INTERFACE Iterator

METHOD current : Object
VAR_INPUT
END_VAR
END_METHOD

METHOD hasNext : BOOL
VAR_INPUT
END_VAR
END_METHOD

METHOD next : Object
VAR_INPUT
END_VAR
END_METHOD

PROPERTY Position : INT
GET
END_GET
END_PROPERTY

METHOD reset : BOOL
VAR_INPUT
END_VAR
END_METHOD

END_INTERFACE

(* stored: Version 1.1.0.1, ProductVersion 3.1.4024.12
   Itf Iterator: Id {11e57a1b-5b87-41c6-8866-dab19c5cc778}
   Method current: Id {d60b1888-45a1-4719-b843-c166d488b64a}
   Method hasNext: Id {6e2d7f23-86d9-421b-a328-b7469453c32f}
   Method next: Id {a0f9df8b-6678-45f8-a11d-40ecbf79b0f8}
   Property Position: Id {b2d58fb3-5dc1-4b10-b185-0b3038c26065}
   Get Get: Id {35a09d46-efa2-4701-858c-533b3fd2a835}
   Method reset: Id {3bba04f1-b69f-4a12-a25c-d55f8c90a503} *)
